FUNCTION_BLOCK FB_Actuator IMPLEMENTS I_Actuator
VAR_INPUT
END_VAR
VAR_OUTPUT
END_VAR
VAR
	doValveExtend AT %Q*	: BOOL;
	doValveRetract AT %Q*	: BOOL;
	diRetracted AT %I*		: BOOL;
	diExtended AT %I*		: BOOL;
	ExtendTon				: TON := (PT := T#5S);
	RetractTon				: TON := (PT := T#5S);
	fbExtendAlarm			: FB_TcAlarm;
	fbRetractAlarm			: FB_TcAlarm;
END_VAR

PROPERTY Error : BOOL
GET
END_GET
SET
END_SET
END_PROPERTY

METHOD Extend : INT
VAR_INPUT
END_VAR
Extend := 0;
doValveExtend := TRUE;
doValveRetract := FALSE;
ExtendTon(IN := NOT diExtended);
IF diExtended THEN
	ExtendTon(IN := FALSE);
	IF fbExtendAlarm.bRaised THEN
		fbExtendAlarm.Clear(0, FALSE);
	END_IF
	Extend := 1;
END_IF
IF ExtendTon.Q THEN
	ExtendTON(IN := FALSE);
	fbExtendAlarm.Raise(0);
	Extend := -1;
END_IF
END_METHOD

METHOD FB_init : BOOL
VAR_INPUT
	bInitRetains : BOOL; // if TRUE, the retain variables are initialized (warm start / cold start)
	bInCopyCode : BOOL;  // if TRUE, the instance afterwards gets moved into the copy code (online change)
END_VAR
IF NOT fbExtendAlarm.EqualsToEventEntryEx(stOther := TC_EVENTS.SlitterEvents.ZActuatorExtendError) THEN
	fbExtendAlarm.CreateEx(TC_EVENTS.SlitterEvents.ZActuatorExtendError, FALSE, 0);
END_IF
IF NOT fbRetractAlarm.EqualsToEventEntryEx(stOther := TC_EVENTS.SlitterEvents.ZActuatorRetractError) THEN
	fbRetractAlarm.CreateEx(TC_EVENTS.SlitterEvents.ZActuatorRetractError, FALSE, 0);
END_IF
END_METHOD

PROPERTY IsExtended : BOOL
GET
IsExtended := diExtended;
END_GET
END_PROPERTY

PROPERTY IsRetracted : BOOL
GET
IsRetracted := diRetracted;
END_GET
END_PROPERTY

METHOD Neutral : BOOL
VAR_INPUT
END_VAR
doValveExtend := FALSE;
doValveRetract := FALSE;
Neutral := TRUE;
END_METHOD

METHOD Reset : BOOL
VAR_INPUT
END_VAR
IF fbExtendAlarm.bRaised THEN
	fbExtendAlarm.Clear(0, FALSE);
END_IF
IF fbRetractAlarm.bRaised THEN
	fbRetractAlarm.Clear(0, FALSE);
END_IF
ExtendTon(IN := FALSE);
RetractTon(IN := FALSE);
END_METHOD

METHOD Retract : INT
VAR_INPUT
END_VAR
Retract := 0;
doValveExtend := FALSE;
doValveRetract := TRUE;
RetractTon(IN := NOT diRetracted);
IF diRetracted THEN
	RetractTon(IN := FALSE);
	IF fbRetractAlarm.bRaised THEN
		fbRetractAlarm.Clear(0, FALSE);
	END_IF
	Retract := 1;
END_IF
IF RetractTon.Q THEN
	RetractTon(IN := FALSE);
	fbRetractAlarm.Raise(0);
	Retract := -1;
END_IF
END_METHOD

END_FUNCTION_BLOCK

(* stored: Version 1.1.0.1, ProductVersion 3.1.4024.9
   POU FB_Actuator: Id {857ac5c9-f12a-4ec3-ab61-971035c91f49}, SpecialFunc None
   Property Error: Id {ec55e1c0-68f0-45f4-abfe-296dc5842a30}
   Get Get: Id {0776e14e-e53f-4b46-858c-5b0950c917c4}
   Set Set: Id {2fee1fbc-8e09-450a-9794-4f5a34adbd41}
   Method Extend: Id {857b4b7c-a2d9-4361-af63-b50945009eef}
   Method FB_init: Id {d803e1fd-381b-411d-9c01-017ca78e6148}
   Property IsExtended: Id {3ecf1009-558a-476e-a119-1f70eca85299}
   Get Get: Id {238dc25c-d1de-4ba0-a529-793e2fe7a545}
   Property IsRetracted: Id {445c5812-266f-4e32-98d0-158014a88419}
   Get Get: Id {e66c6bb5-a345-4806-8914-f5d564d153d0}
   Method Neutral: Id {30b3120a-4bee-44b3-9103-f4dc02b9c992}
   Method Reset: Id {3043bb29-efa2-4f3f-b085-076ab0c786a4}
   Method Retract: Id {d45c1924-cbea-414e-9d60-745d4b4de82d} *)
